FUNCTION RANGE_TO_BYTE : BYTE
VAR_INPUT
	X : REAL;
	low : REAL;
	high : REAL;
END_VAR


(*
version 1.0	9. jan 2008
programmer 	hugo
tested by		tobias

Range_to_byte converts a real value between low and high into a byte

*)

RANGE_TO_BYTE := INT_TO_BYTE(TRUNC_INT((LIMIT(low, X, high) - low) * 255.0 / (high - low)));


(* revision history
hm	9. jan 2008		rev 1.0
	original version

*)

END_FUNCTION

(* stored: Version 1.1.0.1, ProductVersion 3.1.4022.7
   POU RANGE_TO_BYTE: Id {8dc4df7e-933b-4022-94ac-ebe520dff073}, SpecialFunc None *)
